{attribute 'qualified_only'}
VAR_GLOBAL
	aTaskInfo							: ARRAY[1..SIZEOF(TwinCAT_SystemInfoVarList._TaskInfo)/SIZEOF(PlcTaskSystemInfo)] OF ST_Log4TcTaskInfo;
END_VAR

(* stored: Version 1.1.0.1, ProductVersion 3.1.4024.0
   GVL Log4TcInfo: Id {9ec35cf4-7760-4c91-99dd-d77cc6c9acf2} *)
